PROGRAM MAIN
VAR
END_VAR

END_PROGRAM

(* stored: Version 1.1.0.1
   POU MAIN: Id {a0eda2ac-34e9-4306-912e-fa92d32909de} *)
